TYPE ST_Alarm :
STRUCT
    bCondition      : BOOL;           
    nID             : UDINT;           
    nSeverity       : UINT;     
	sMessage        : STRING(255);        
END_STRUCT
END_TYPE

(* stored: Version 1.1.0.1, ProductVersion 3.1.4026.11
   DUT ST_Alarm: Id {62903e3f-1b71-43bd-bca3-90f8ae946812} *)
